(* Logix 5000 project; controller Animation_With_Max_And_Min_Range Emulate 5570 rev 30.12; software revision 30.01 *)

TASK MainTask (continuous, watchdog 500 ms) : MainProgram

MODULES
   Local : Emulate 5570 (ICP 2, rev 30.12)
END_MODULES

PROGRAM MainProgram   (* main routine MainRoutine *)
VAR
   Delay : TIMER;
   Fill : BOOL;
   Min : DINT;
   Power : BOOL;
   Start : BOOL;
   Stop : BOOL;
END_VAR

ROUTINE MainRoutine   (* ladder *)
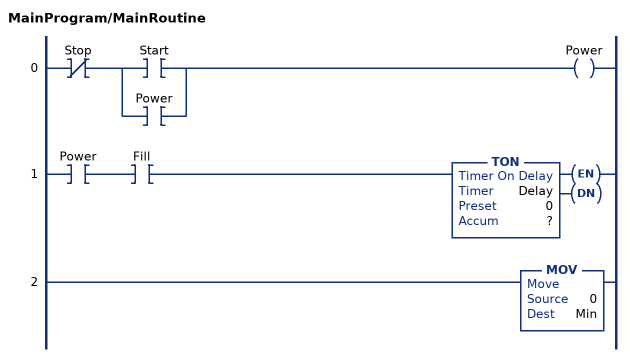
   0: XIO(Stop)[XIC(Start) ,XIC(Power) ]OTE(Power);
   1: XIC(Power)XIC(Fill)TON(Delay,?,?);
   2: MOV(0,Min);
END_ROUTINE
END_PROGRAM
